// TIA Portal V15.1 export
// export: Created 2025-12-09T12:22:57.8982402Z, ExportSetting WithDefaults, WithReadOnly, DisplayName Totally Integrated Automation Portal, DisplayVersion V15.1, DisplayName TIA Portal Openness, DisplayVersion V15.1, DisplayName SINAMICS Startdrive Advanced, DisplayVersion V15.1, DisplayName SINAMICS DCC, DisplayVersion V15.1, DisplayName G130, G150, S120, S150, SINAMICS MV, S210, DisplayVersion V15.1, DisplayName G110M, G120, G120C, G120D, G120P, DisplayVersion V15.1, DisplayName STEP 7 Professional, DisplayVersion V15.1, DisplayName STEP 7 Safety, DisplayVersion V15.1, DisplayName WinCC Professional, DisplayVersion V15.1, DisplayName SIMATIC Visualization Architect, DisplayVersion V15.1
DATA_BLOCK "[nome_robo]#FB_Rob_PN_E_DB"   // DB[numero_db]
{ S7_Optimized_Access := 'TRUE' }
AUTHOR : VASS_V05
FAMILY : ROBPNE
VERSION : 0.0
// Eingänge Roboter
// stored: AutoNumber false, CodeModifiedDate 2018-07-12T14:46:14.8740198Z, CompileDate 2019-04-01T14:36:11.5725261Z, CreationDate 2017-04-11T19:23:05.038059Z, DBAccessibleFromOPCUA true, DownloadWithoutReinit false, InstanceOfName FB_Rob_PN_E, InstanceOfNumber 202, InstanceOfType FB, InterfaceModifiedDate 2018-07-06T08:52:26.862081Z, IsConsistent true, IsKnowHowProtected false, IsRetainMemResEnabled false, MemoryReserve 100, ModifiedDate 2018-07-12T14:46:14.8740198Z, ParameterModified 2018-03-22T07:53:41.5036336Z, StructureModified 2018-04-03T10:13:14.1811337Z, UDAEnableTagReadback false
"FB_Rob_PN_E"
   // VAR_IN_OUT
   //    Rob_E : "ST_Rob_E";
   //    ST_ROB : "ST_Rob";
   // END_VAR
   // VAR
   //    diPOS_BLK { ExternalAccessible := 'False'; ExternalVisible := 'False'; ExternalWritable := 'False'} : DInt;
   //    "255" { ExternalAccessible := 'False'; ExternalVisible := 'False'; ExternalWritable := 'False'} : Bool;
   // END_VAR
BEGIN
END_DATA_BLOCK
